// TwinCAT 3 PLC project Test1
// ProgramVersion: 3.1.4023.0
// libraries:
//   Tc2_Standard, * (Beckhoff Automation GmbH)
//   Tc2_System, * (Beckhoff Automation GmbH)
//   Tc3_IotBase, * (Beckhoff Automation GmbH)
//   Tc3_Module, * (Beckhoff Automation GmbH)
// project tree:
//   / MQTTTask.TcTTO, PlcTask.TcTTO
//   POUs/ MAIN.TcPOU, MQTT_MAIN.TcPOU
// real-time tasks:
//   TASK PlcTask: cycle T#1000ms, priority 20, ADS port 350
//   TASK MQTTTask: cycle T#10ms, priority 21, ADS port 351

CONFIGURATION Test1
    RESOURCE PLC ON TwinCAT3
        TASK MQTTTask(INTERVAL := T#10ms, PRIORITY := 21);
        TASK PlcTask(INTERVAL := T#1000ms, PRIORITY := 20);
        PROGRAM MQTT_MAIN WITH MQTTTask : MQTT_MAIN;
        PROGRAM MAIN WITH PlcTask : MAIN;
    END_RESOURCE
END_CONFIGURATION

// ---- POUs/MQTT_MAIN.TcPOU
PROGRAM MQTT_MAIN
VAR
	fbMqttClient : FB_IotMqttClient;
	bSetParmeter : BOOL := TRUE;
	bconnect : BOOL := TRUE;
	
	sTopicPub1 : STRING := 'my first topic';
	sTopicPub2 : STRING := 'my second topic'; 
	sPayloadPub : STRING;
	i : UINT;
	fbTimer : TON := (PT:=T#1S);
	
	bSubscribed : BOOL;
	//sTopicSub : STRING := 'topic';
	//sTopicRcv : STRING;
	sPayloadRcv1 : STRING(255);
    sPayloadRcv2 : STRING(255);
	fbMessageQueue : FB_IotMqttMessageQueue;
	fbMessage : FB_IotMqttMessage;

	//nPayloadSize : UDINT;

END_VAR
VAR CONSTANT
    (* subscriptions *)
    sTopicSub1 : STRING(255) := 'my first topic';
    sTopicSub2 : STRING(255) := 'my second topic'; 
END_VAR

IF bSetParmeter THEN
	bSetParmeter := FALSE;
	fbMqttClient.sHostName := '192.168.0.144';
	fbMqttClient.nHostPort := 1883;
	fbMqttClient.sTopicPrefix := '';
	fbMqttClient.ipMessageQueue := fbMessageQueue;
	
END_IF

fbMqttClient.Execute(bconnect);


IF fbMqttClient.bConnected THEN
	IF NOT bSubscribed THEN
		bSubscribed := fbMqttClient.Subscribe(sTopic := sTopicSub1, eQos := TcIotMqttQos.AtMostOnceDelivery);
		bSubscribed := fbMqttClient.Subscribe(sTopic := sTopicSub2, eQos := TcIotMqttQos.AtMostOnceDelivery);
	END_IF
	fbTimer(IN:=TRUE);
	IF fbTimer.Q THEN
		fbTimer(IN :=FALSE);
		i := i+1;
		IF i MOD 2 = 1 THEN
			sPayloadPub := CONCAT('MyMessage', TO_STRING(i));
			fbMqttClient.Publish( sTopic:= sTopicPub1, pPayload := ADR(sPayloadPub), nPayloadSize := SIZEOF(sPayloadPub)+1, 
							eQoS := TcIotMqttQos.AtMostOnceDelivery, bRetain:= FALSE, bQueue := FALSE);
		ELSE
			sPayloadPub := CONCAT('MyMessage', TO_STRING(i));
			fbMqttClient.Publish( sTopic:= sTopicPub2, pPayload := ADR(sPayloadPub), nPayloadSize := SIZEOF(sPayloadPub)+1, 
							eQoS := TcIotMqttQos.AtMostOnceDelivery, bRetain:= FALSE, bQueue := FALSE);
		END_IF
	END_IF
	
END_IF
IF fbMessageQueue.nQueuedMessages > 0 THEN
    IF fbMessageQueue.Dequeue(fbMessage:=fbMessage) THEN
        IF fbMessage.CompareTopic(sTopic:=sTopicSub1) THEN
            fbMessage.GetPayload(pPayload:=ADR(sPayloadRcv1), nPayloadSize:=SIZEOF(sPayloadRcv1), bSetNullTermination:=FALSE);
        ELSIF fbMessage.CompareTopic(sTopic:=sTopicSub2) THEN
            fbMessage.GetPayload(pPayload:=ADR(sPayloadRcv2), nPayloadSize:=SIZEOF(sPayloadRcv2), bSetNullTermination:=FALSE);
        END_IF
    END_IF
END_IF

END_PROGRAM

// ---- POUs/MAIN.TcPOU
PROGRAM MAIN
VAR
	a : UINT;
	b : UINT;
	c : UINT;
	x : UINT;
	y : UINT;
	i : UINT;
	j : UINT;
	k : UINT;
	q : UINT;
	w : UINT;
	e : UINT;
	
	
	
	bInit :	BOOL;
	
	bTRUE : BOOL;
END_VAR

a := a+1;
IF a = 10 THEN 
	FOR a := 1 TO 10 DO
		c := c + 1;
	END_FOR
END_IF

(*IF a = 10 THEN
	c := 0;
END_IF

FOR a := 1 TO 10 BY 1 DO
	c := c + 1;
END_FOR

CASE b OF
	1 :
	a := 1;
	2:
	b := 2;
	3:
	c := 3;
	4:
	a := 0;
	
END_CASE*)

END_PROGRAM
